FUNCTION_BLOCK EL5072
VAR
	_io : EL5072_Data;
	{attribute addProperty Name "WcState"}
	_wcState : WcStateInputToggle;
	{attribute addProperty Name "Info data"}
	_infoData : InfoDataAdsDC;
END_VAR

PROPERTY IO : REFERENCE TO EL5072_Data
GET
IO REF= _io;
END_GET
END_PROPERTY

PROPERTY WcState : REFERENCE TO WcStateInputToggle
GET
WcState REF= _wcState;
END_GET
END_PROPERTY

END_FUNCTION_BLOCK

(* stored: Version 1.1.0.1, ProductVersion 3.1.4024.9
   POU EL5072: Id {661530b7-05b4-0e2b-1f62-4917b3477550}, SpecialFunc None
   Property IO: Id {6b4da506-4d68-0203-3f0e-3d4ac373a747}
   Get Get: Id {093d218f-2306-0433-1c6e-e96dfb761d0c}
   Property WcState: Id {f46b6aa1-d311-0c8b-0754-4f1292f40484}
   Get Get: Id {5eff771d-076a-0e7e-0ced-5c120f7a2343} *)
